# EPICS autosave request: GalilSup/Db/GALIL_controller_kinematics.req
# Kinematics

# Forward transforms (Readbacks)
file "galil_forward_transform.req" P=$(P), M=MTR$(CCP)09
file "galil_forward_transform.req" P=$(P), M=MTR$(CCP)10
file "galil_forward_transform.req" P=$(P), M=MTR$(CCP)11
file "galil_forward_transform.req" P=$(P), M=MTR$(CCP)12
file "galil_forward_transform.req" P=$(P), M=MTR$(CCP)13
file "galil_forward_transform.req" P=$(P), M=MTR$(CCP)14
file "galil_forward_transform.req" P=$(P), M=MTR$(CCP)15
file "galil_forward_transform.req" P=$(P), M=MTR$(CCP)16

# Reverse transforms (Setpoints)
file "galil_reverse_transforms.req" P=$(P), M=MTR$(CCP)09
file "galil_reverse_transforms.req" P=$(P), M=MTR$(CCP)10
file "galil_reverse_transforms.req" P=$(P), M=MTR$(CCP)11
file "galil_reverse_transforms.req" P=$(P), M=MTR$(CCP)12
file "galil_reverse_transforms.req" P=$(P), M=MTR$(CCP)13
file "galil_reverse_transforms.req" P=$(P), M=MTR$(CCP)14
file "galil_reverse_transforms.req" P=$(P), M=MTR$(CCP)15
file "galil_reverse_transforms.req" P=$(P), M=MTR$(CCP)16
